FUNCTION_BLOCK E_PULSE (* standard timer function block (pulse) *)
  (* Standard: 61499-2; Description: Copyright (c) 2023, 2024 HR Agrartechnik GmbH This program and the accompanying materials are made available under the terms of the Eclipse Public License 2.0 which is available at https://www.eclipse.org/legal/epl-2.0/ SPDX-License-Identifier: EPL-2.0  This FB makes a Impulse of Duration TM on the Output QO. *)
  (* Version 1.0, 2023-08-21, Franz Hoepfinger, HR Agrartechnik GmbH, initial implementation as E_IMPULSE *)
  (* Version 1.0, 2024-03-05, Franz Hoepfinger, HR Agrartechnik GmbH, renamed to E_PULSE *)
  (* Version 1.1, 2024-04-23, Franz Hoepfinger, HR Agrartechnik GmbH, Add a Reset to Timer FBs *)
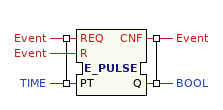
  EVENT_INPUT
    REQ WITH PT; (* Service Request *)
    R; (* Reset *)
  END_EVENT
  EVENT_OUTPUT
    CNF WITH Q; (* Confirmation of Requested Service *)
  END_EVENT
  VAR_INPUT
    PT : TIME; (* Pulse time *)
  END_VAR
  VAR_OUTPUT
    Q : BOOL; (* Output *)
  END_VAR
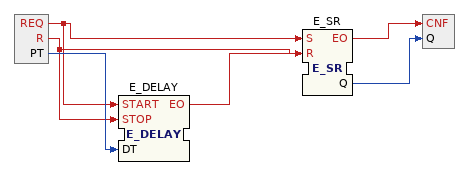
  FBS
    E_DELAY : E_DELAY;
    E_SR : E_SR;
  END_FBS
  EVENT_CONNECTIONS
    REQ TO E_DELAY.START;
    REQ TO E_SR.S;
    E_DELAY.EO TO E_SR.R;
    E_SR.EO TO CNF;
    R TO E_DELAY.STOP;
    R TO E_SR.R;
  END_CONNECTIONS
  DATA_CONNECTIONS
    PT TO E_DELAY.DT;
    E_SR.Q TO Q;
  END_CONNECTIONS
END_FUNCTION_BLOCK
